Fanuc KAREL source: KD00019.KL

PROGRAM KD00019
%NOLOCKGROUP
TYPE
  REC_T = STRUCTURE
    VALUE: INTEGER
  ENDSTRUCTURE
VAR
  I: INTEGER
  J: INTEGER
  B: BOOLEAN
  R: REAL
  S: STRING[80]
  REC: REC_T
BEGIN
  REC.VALUE = 1
  USING REC DO
    VALUE = VALUE + 1
  ENDUSING
END KD00019
